{attribute 'qualified_only'}
VAR_GLOBAL
END_VAR

(* stored: Version 1.1.0.1, ProductVersion 3.1.4022.7
   GVL GVL_01_Function: Id {75f84da1-b551-42ec-b2ec-652849371723} *)
